VISUALIZATION Page_2  // 2x2
END_VISUALIZATION

(* stored: Version 1.1.0.1, ProductVersion 3.1.4024.12
   Visu Page_2: Id {ba727a93-1bf6-4856-bfb8-6a64a90ef92e} *)
